// Mitsubishi GX Works2 project: Project   PLC: FX3G

// global labels: Global1
VAR_GLOBAL
  startDay AT X007 : BOOL;
  stillOpen AT Y007 : BOOL;
  Click_X5 AT X005 : BOOL;
  Analog_Output AT D8282 : INT;
  Analog_Input1 AT D8280 : INT;
  raspberryInentory AT D1111 : REAL;
  lemonInentory AT D2222 : REAL;
  stabilizerInentory AT D3333 : REAL;
  gummyBearsInentory AT D4444 : REAL;
  raspberryIceCreamRegular : REAL;
  raspberryIceCreamTreat : REAL;
  lemonIceCreamRegular : REAL;
  lemonIceCreamTreat : REAL;
  raspberryIceCreamContainer : REAL;
  lemonIceCreamContainer : REAL;
  coolingContainerRasp : REAL;
  coolingContainerLemon : REAL;
  mixContainer : REAL;
  startIceCreaming AT X001 : BOOL;
END_VAR
VAR_GLOBAL CONSTANT
  normalization : REAL := E400;
  ifLessThan10 : REAL := E10;
END_VAR
VAR_GLOBAL
  isRegular AT M1 : BOOL;
  isTreat AT M2 : BOOL;
END_VAR
VAR_GLOBAL CONSTANT
  rasbNeededRegular : REAL := E280.0;
  lemonNeededRegular : REAL := E455.0;
  stabNeededRegular : REAL := E105.0;
  bearNeededRegular : REAL := E28.0;
  rasbNeededTreat : REAL := E385.0;
  lemonNeededTreat : REAL := E665.0;
  stabNeededTreat : REAL := E210.0;
  bearNeededTreat : REAL := E70.0;
END_VAR
VAR_GLOBAL
  isRegPossible AT M3 : BOOL;
  isTreatPossible AT M4 : BOOL;
  FinishRegularToday AT M15 : BOOL;
  FinishTreatToday AT M16 : BOOL;
  StillPossible AT M50 : BOOL;
  FisrtStageIceCreamingReg AT M5 : BOOL;
  FisrtStageIceCreamingTreat AT M6 : BOOL;
  iceCreamDuration AT Y000 : BOOL;
  TimeCoil AT TC1 : BOOL;
  FiveSec AT K50 : INT;
  TimerWhileIceCreaming AT TS1 : BOOL;
END_VAR
VAR_GLOBAL CONSTANT
  raspberryIceCreamAddReg : REAL := E350.0;
  lemonIceCreamAddReg : REAL := E490.0;
  raspberryIceCreamAddTreat : REAL := E560.0;
  lemonIceCreamAddTreat : REAL := E700.0;
END_VAR
VAR_GLOBAL
  Sen_10 AT X003 : BOOL;
  TransferIceCream AT X002 : BOOL;
  LightForCooling AT Y002 : BOOL;
  TimerWhileCooling AT TC2 : BOOL;
  EightSec AT K80 : INT;
  TimerWhileCoolings AT TS2 : BOOL;
  MixRegular AT M51 : BOOL;
  MixTreat AT M61 : BOOL;
  WhileMixing_1 AT Y005 : BOOL;
  M_46 AT M46 : BOOL;
  startBlink5 AT TC50 : BOOL;
  MixingRegular AT TC30 : BOOL;
  MixingReg AT K30 : INT;
  MixingTreat AT TC55 : BOOL;
  DoneMixingRegular AT TS30 : BOOL;
  DoneMixingTreat AT TS55 : BOOL;
  Blink AT K5 : INT;
  ifEnoughBearRegular AT M7 : BOOL;
  ifEnoughBearTreat AT M8 : BOOL;
  Y5_Blinking AT TS50 : BOOL;
  startBlink6 AT TC60 : BOOL;
  Y6_Blinking AT TS60 : BOOL;
  WhileMixing_2 AT Y006 : BOOL;
  Pack1gumigum AT X000 : BOOL;
  IndicatorForX0 AT M20 : BOOL;
  cc1 AT CC1 : BOOL;
  startPacking AT X004 : BOOL;
  FirstGumigumInPackage AT Y004 : BOOL;
  GumigumPackage AT CS1 : BOOL;
  CounterGummies_7 AT K7 : INT;
  stillPacking AT M80 : BOOL;
  NumOfGummygamPacks AT D8284 : REAL;
END_VAR
VAR_GLOBAL CONSTANT
  AddPack : REAL := E0.01;
  MulConst : REAL := E4000.0;
  bearsForReg : REAL := E28.0;
  bearsForTreat : REAL := E70.0;
END_VAR
VAR_GLOBAL
  storageContainer : REAL;
END_VAR
VAR_GLOBAL CONSTANT
  storageCounter : REAL := E1.0;
  regularAmount : REAL := E868;
  treatAmount : REAL := E1330;
  ifGreaterThan6 : REAL := E6;
  ifBetween0_5 : REAL := E5;
  reset : REAL := E0.0;
END_VAR
VAR_GLOBAL
  finishedIteration AT M100 : BOOL;
  ifDone AT M200 : BOOL;
END_VAR

// task Task_01 (event TRUE, interval 0, priority 31): POU_01

PROGRAM POU_01
(* structured ladder/FBD written out as ST: instructions are called as NAME(EN, inputs, outputs); _pN, _eN, _tN stand for wires *)
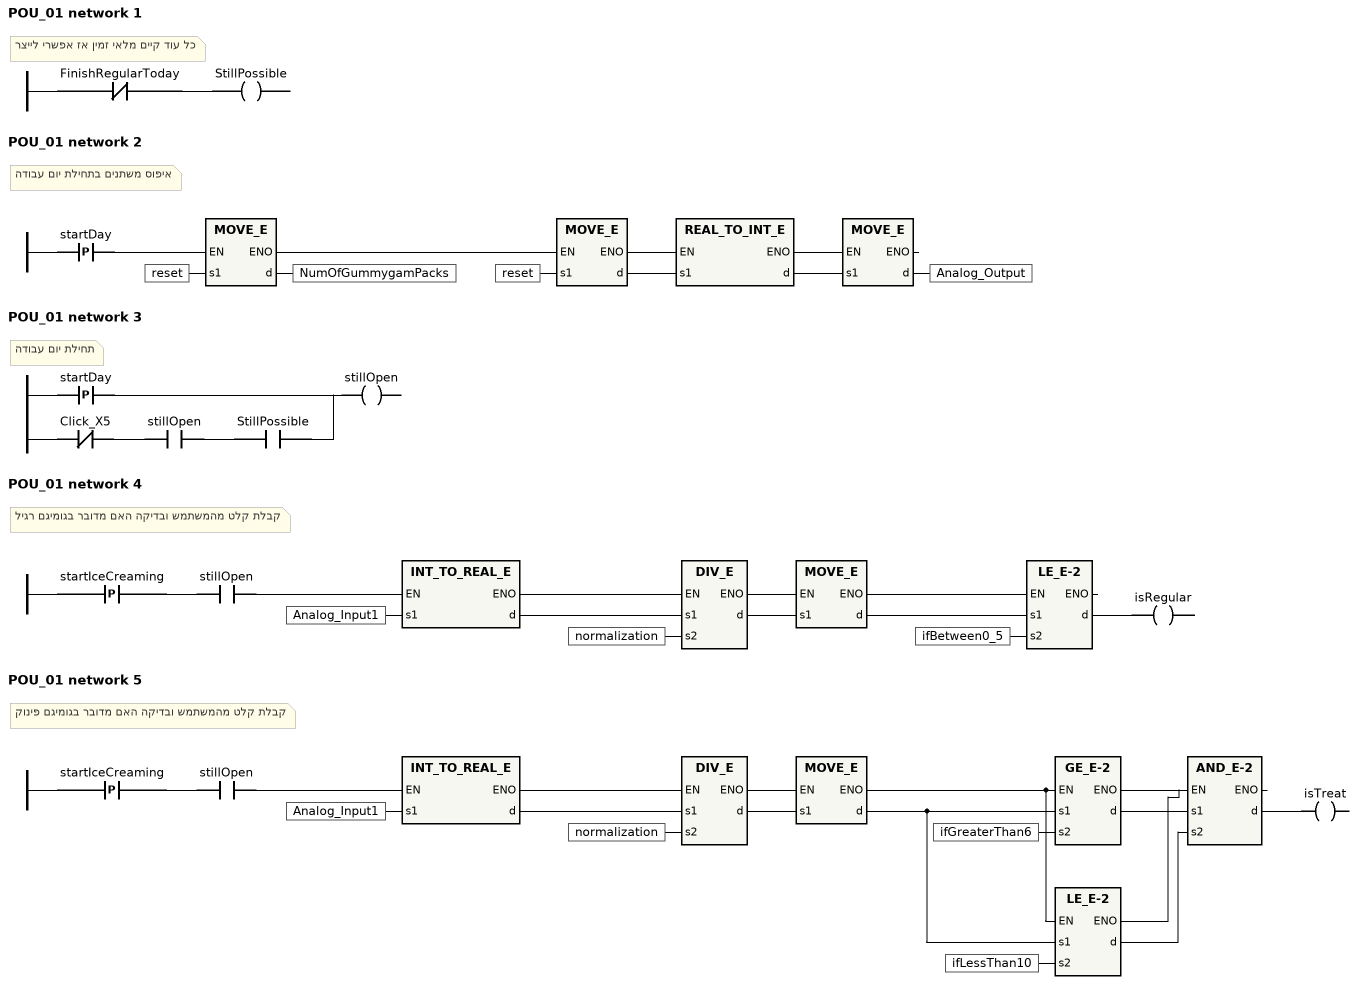
(* network 1 *)
(* כל עוד קיים מלאי זמין אז אפשרי לייצר *)
StillPossible := NOT FinishRegularToday;
(* network 2 *)
(* איפוס משתנים בתחילת יום עבודה *)
_e1 := MOVE_E(LDP(TRUE, startDay), reset, NumOfGummygamPacks);
_e3 := MOVE_E(_e1, reset, _t2);
_e5 := REAL_TO_INT_E(_e3, _t2, _t4);
MOVE_E(_e5, _t4, Analog_Output);
(* network 3 *)
(* תחילת יום עבודה *)
stillOpen := LDP(TRUE, startDay) OR (NOT Click_X5 AND stillOpen AND StillPossible);
(* network 4 *)
(* קבלת קלט מהמשתמש ובדיקה האם מדובר בגומיגם רגיל *)
_e2 := INT_TO_REAL_E(LDP(TRUE, startIceCreaming) AND stillOpen, Analog_Input1, _t1);
_e4 := DIV_E(_e2, _t1, normalization, _t3);
_e6 := MOVE_E(_e4, _t3, _t5);
LE_E(_e6, _t5, ifBetween0_5, _t7);
isRegular := _t7;
(* network 5 *)
(* קבלת קלט מהמשתמש ובדיקה האם מדובר בגומיגם פינוק *)
_e2 := INT_TO_REAL_E(LDP(TRUE, startIceCreaming) AND stillOpen, Analog_Input1, _t1);
_e4 := DIV_E(_e2, _t1, normalization, _t3);
_e6 := MOVE_E(_e4, _t3, _t5);
_e8 := GE_E(_e6, _t5, ifGreaterThan6, _t7);
_e10 := LE_E(_e6, _t5, ifLessThan10, _t9);
AND_E(_e8 OR _e10, _t7, _t9, _t11);
isTreat := _t11;
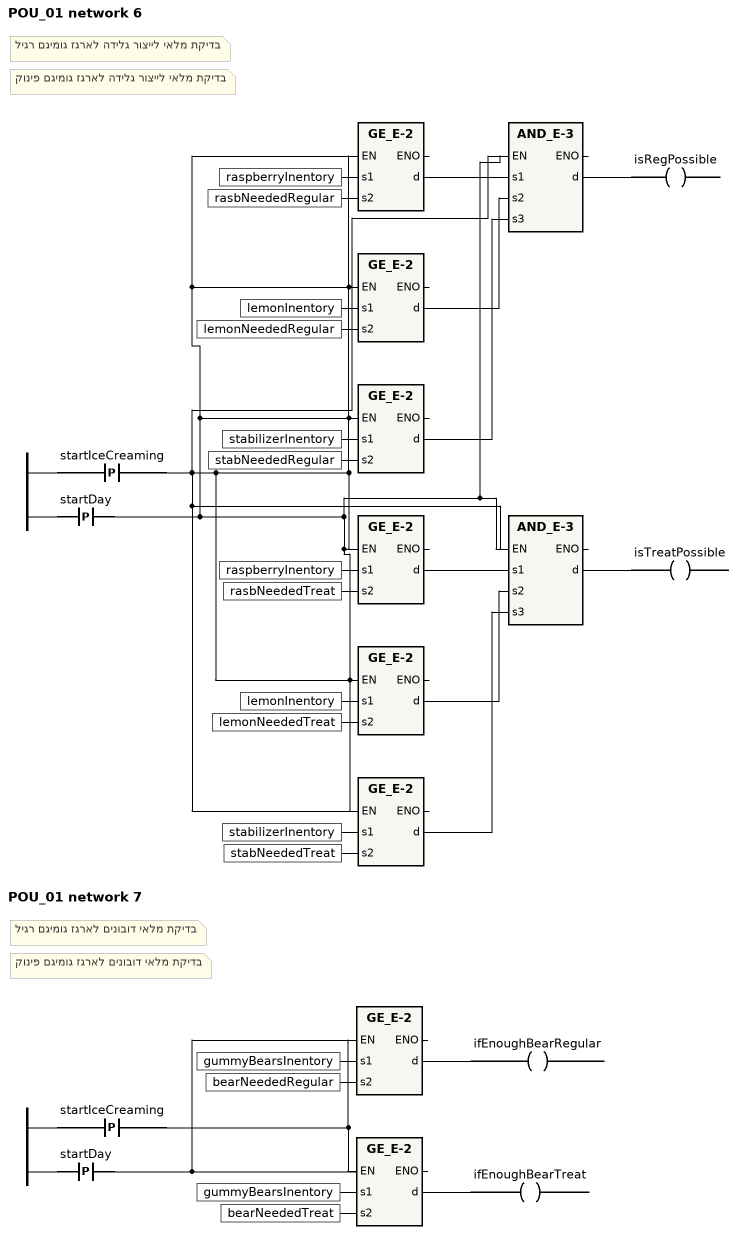
(* network 6 *)
(* בדיקת מלאי לייצור גלידה לארגז גומיגם רגיל *)
(* בדיקת מלאי לייצור גלידה לארגז גומיגם פינוק *)
_p1 := LDP(TRUE, startIceCreaming) OR LDP(TRUE, startDay);
GE_E(_p1, raspberryInentory, rasbNeededRegular, _t2);
GE_E(_p1, lemonInentory, lemonNeededRegular, _t3);
GE_E(_p1, stabilizerInentory, stabNeededRegular, _t4);
AND_E(_p1, _t2, _t3, _t4, _t5);
isRegPossible := _t5;
GE_E(_p1, raspberryInentory, rasbNeededTreat, _t6);
GE_E(_p1, lemonInentory, lemonNeededTreat, _t7);
GE_E(_p1, stabilizerInentory, stabNeededTreat, _t8);
AND_E(_p1, _t6, _t7, _t8, _t9);
isTreatPossible := _t9;
(* network 7 *)
(* בדיקת מלאי דובונים לארגז גומיגם רגיל *)
(* בדיקת מלאי דובונים לארגז גומיגם פינוק *)
_p1 := LDP(TRUE, startIceCreaming) OR LDP(TRUE, startDay);
GE_E(_p1, gummyBearsInentory, bearNeededRegular, _t2);
ifEnoughBearRegular := _t2;
GE_E(_p1, gummyBearsInentory, bearNeededTreat, _t3);
ifEnoughBearTreat := _t3;
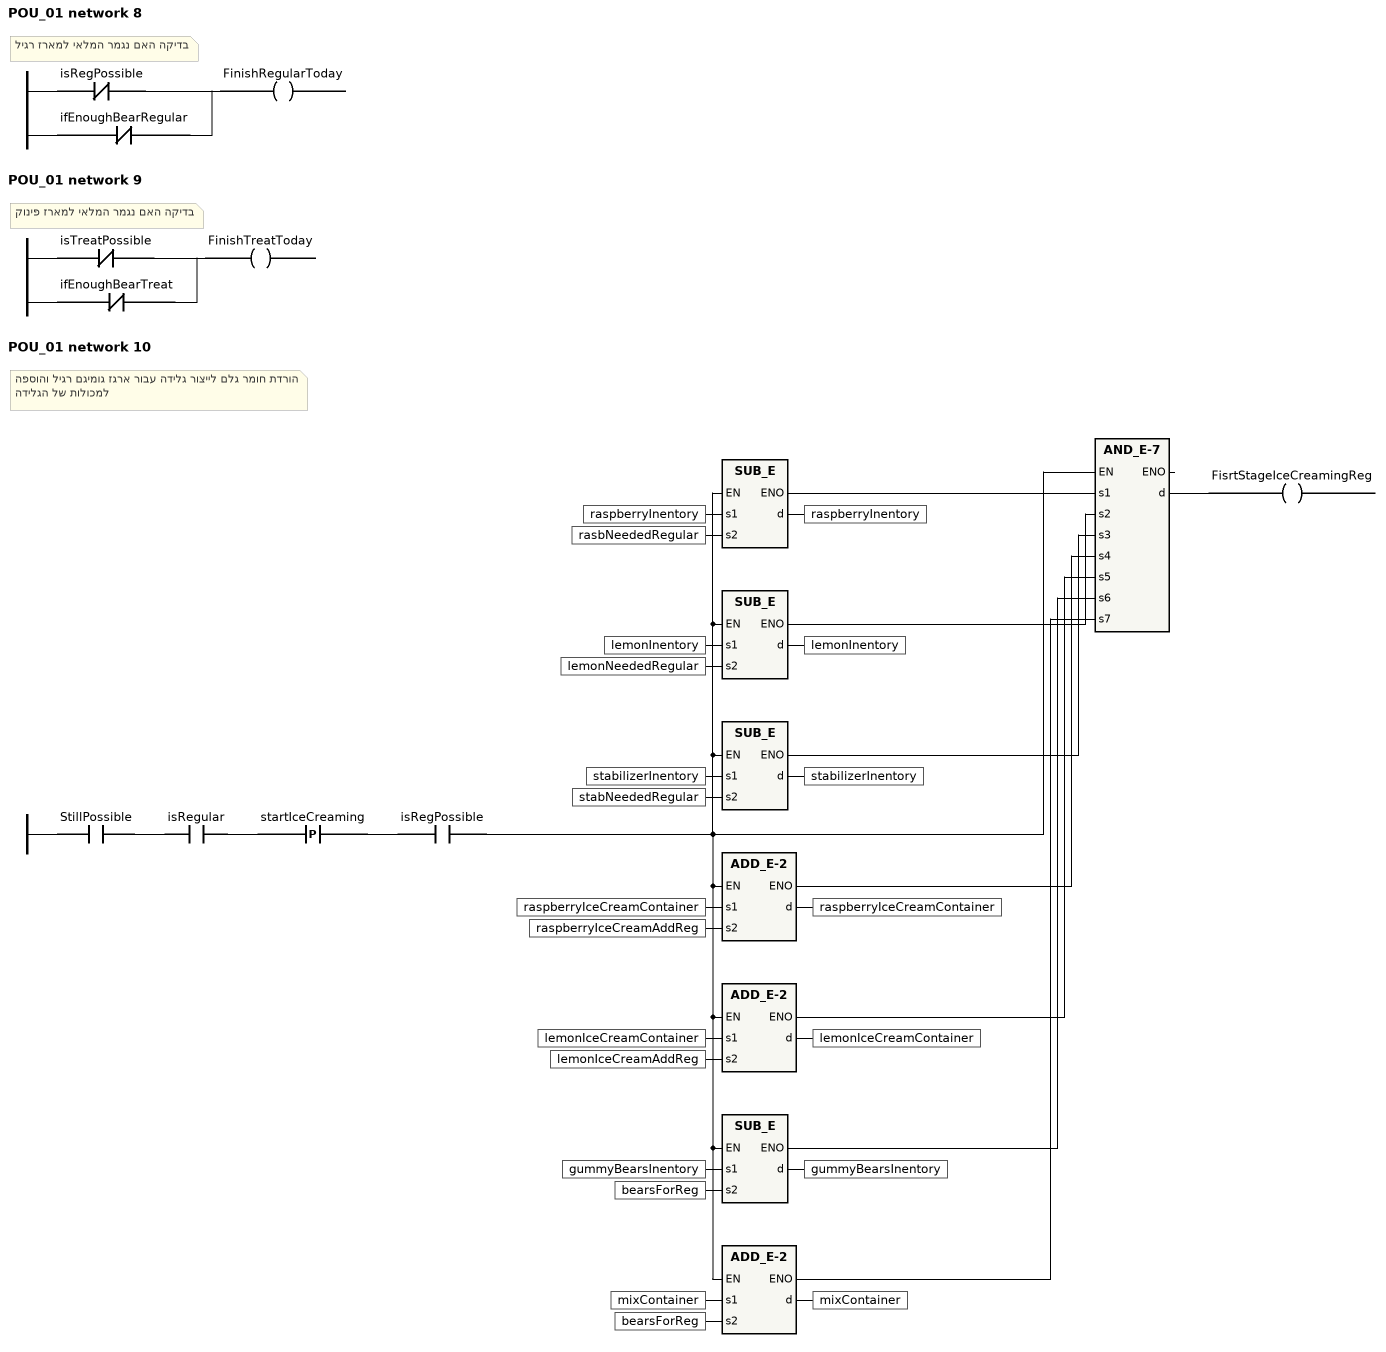
(* network 8 *)
(* בדיקה האם נגמר המלאי למארז רגיל *)
FinishRegularToday := (NOT isRegPossible) OR (NOT ifEnoughBearRegular);
(* network 9 *)
(* בדיקה האם נגמר המלאי למארז פינוק *)
FinishTreatToday := (NOT isTreatPossible) OR (NOT ifEnoughBearTreat);
(* network 10 *)
(* הורדת חומר גלם לייצור גלידה עבור ארגז גומיגם רגיל והוספה למכולות של הגלידה *)
_p1 := StillPossible AND isRegular AND LDP(TRUE, startIceCreaming) AND isRegPossible;
_e2 := SUB_E(_p1, raspberryInentory, rasbNeededRegular, raspberryInentory);
_e3 := SUB_E(_p1, lemonInentory, lemonNeededRegular, lemonInentory);
_e4 := SUB_E(_p1, stabilizerInentory, stabNeededRegular, stabilizerInentory);
_e5 := ADD_E(_p1, raspberryIceCreamContainer, raspberryIceCreamAddReg, raspberryIceCreamContainer);
_e6 := ADD_E(_p1, lemonIceCreamContainer, lemonIceCreamAddReg, lemonIceCreamContainer);
_e7 := SUB_E(_p1, gummyBearsInentory, bearsForReg, gummyBearsInentory);
_e8 := ADD_E(_p1, mixContainer, bearsForReg, mixContainer);
AND_E(_p1, _e2, _e3, _e4, _e5, _e6, _e7, _e8, _t9);
FisrtStageIceCreamingReg := _t9;
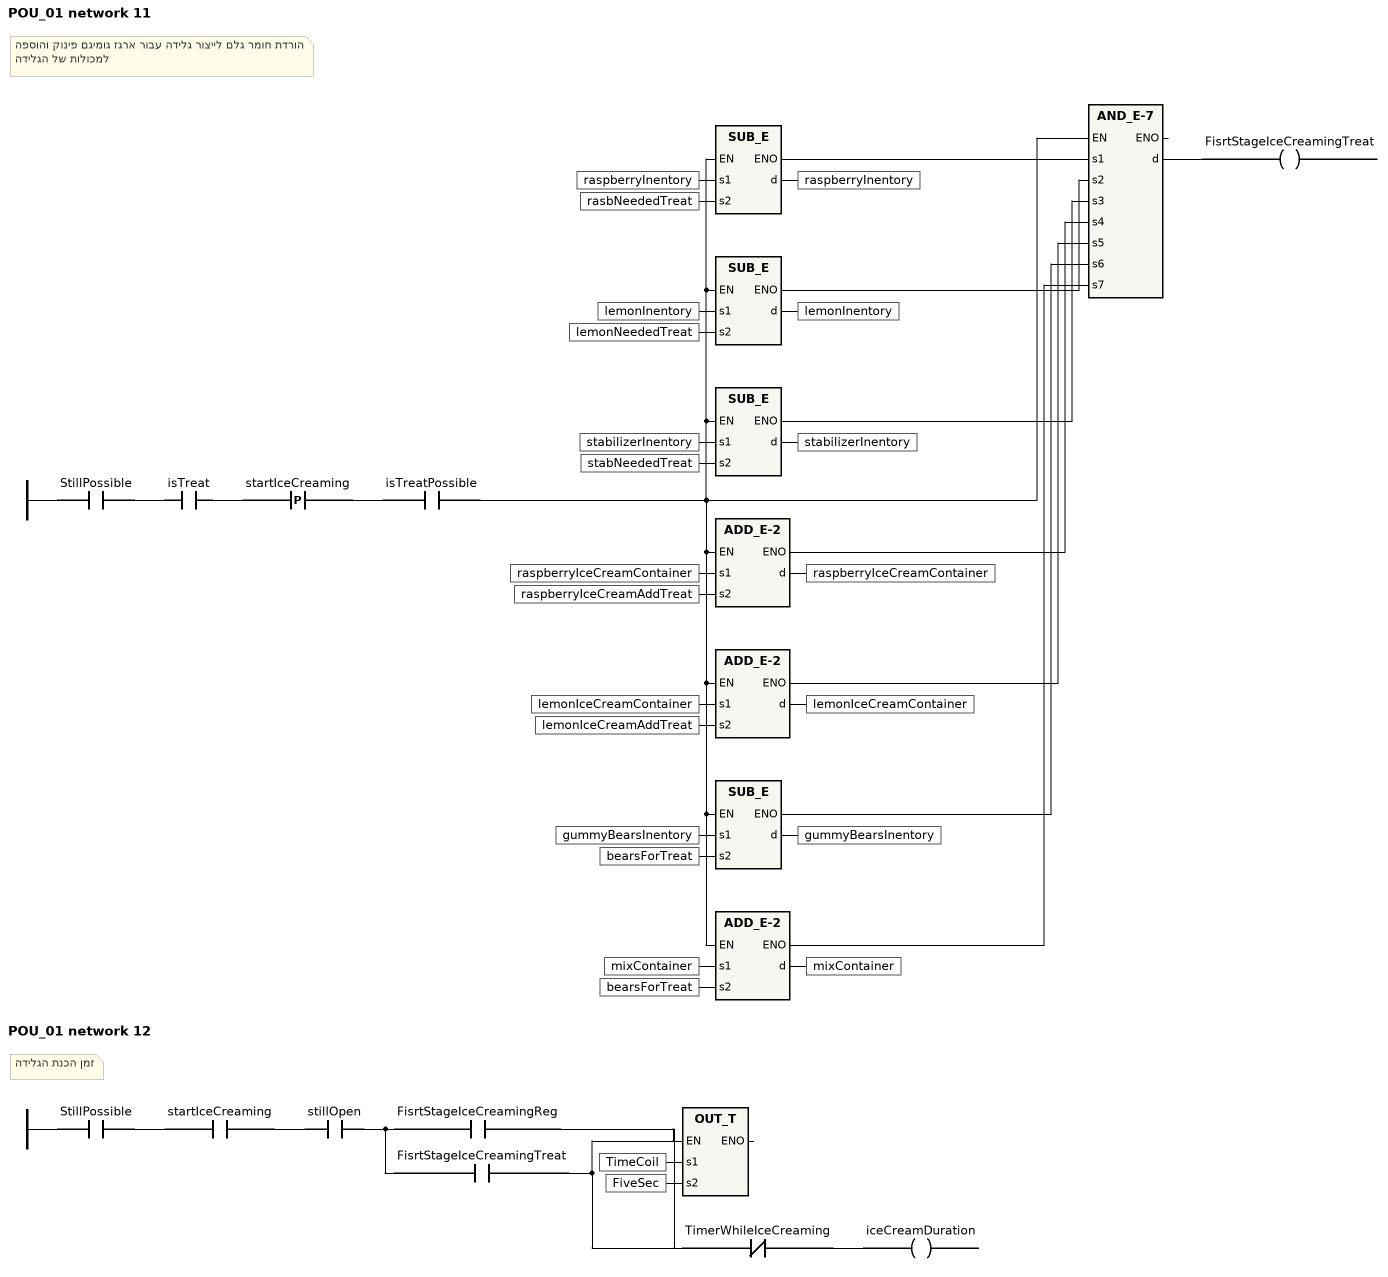
(* network 11 *)
(* הורדת חומר גלם לייצור גלידה עבור ארגז גומיגם פינוק והוספה למכולות של הגלידה *)
_p1 := StillPossible AND isTreat AND LDP(TRUE, startIceCreaming) AND isTreatPossible;
_e2 := SUB_E(_p1, raspberryInentory, rasbNeededTreat, raspberryInentory);
_e3 := SUB_E(_p1, lemonInentory, lemonNeededTreat, lemonInentory);
_e4 := SUB_E(_p1, stabilizerInentory, stabNeededTreat, stabilizerInentory);
_e5 := ADD_E(_p1, raspberryIceCreamContainer, raspberryIceCreamAddTreat, raspberryIceCreamContainer);
_e6 := ADD_E(_p1, lemonIceCreamContainer, lemonIceCreamAddTreat, lemonIceCreamContainer);
_e7 := SUB_E(_p1, gummyBearsInentory, bearsForTreat, gummyBearsInentory);
_e8 := ADD_E(_p1, mixContainer, bearsForTreat, mixContainer);
AND_E(_p1, _e2, _e3, _e4, _e5, _e6, _e7, _e8, _t9);
FisrtStageIceCreamingTreat := _t9;
(* network 12 *)
(* זמן הכנת הגלידה *)
_p1 := StillPossible AND startIceCreaming AND stillOpen;
_p2 := (_p1 AND FisrtStageIceCreamingReg) OR (_p1 AND FisrtStageIceCreamingTreat);
iceCreamDuration := _p2 AND NOT TimerWhileIceCreaming;
OUT_T(_p2, TimeCoil, FiveSec);
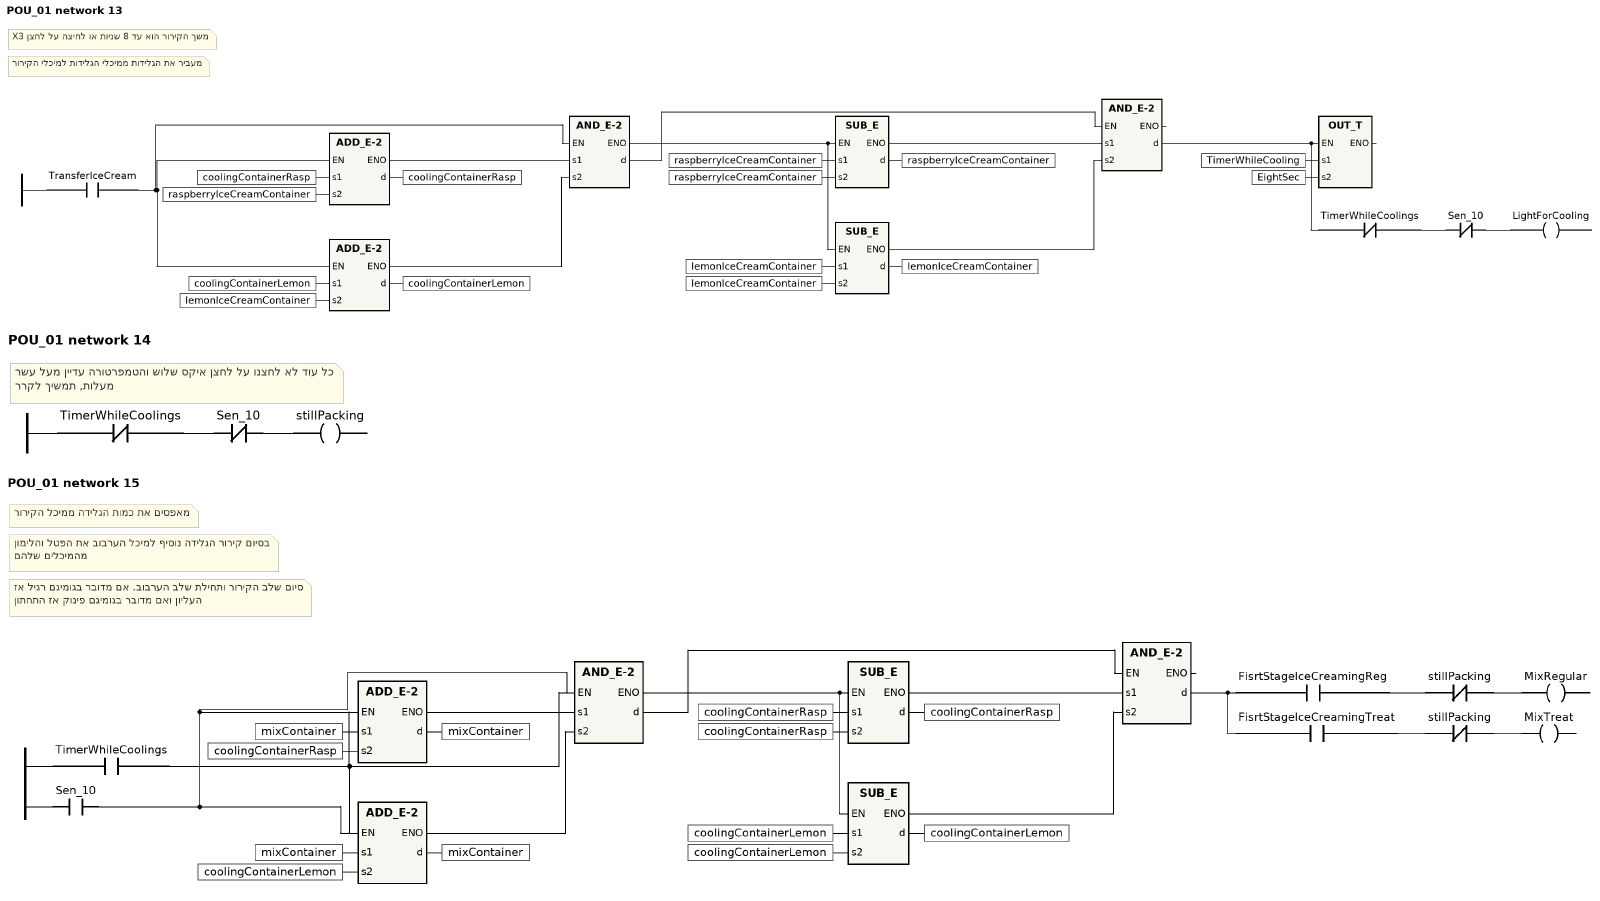
(* network 13 *)
(* משך הקירור הוא עד 8 שניות או לחיצה על לחצן X3 *)
(* מעביר את הגלידות ממיכלי הגלידות למיכלי הקירור *)
_e1 := ADD_E(TransferIceCream, coolingContainerRasp, raspberryIceCreamContainer, coolingContainerRasp);
_e2 := ADD_E(TransferIceCream, coolingContainerLemon, lemonIceCreamContainer, coolingContainerLemon);
_e4 := AND_E(TransferIceCream, _e1, _e2, _t3);
_e5 := SUB_E(_e4, raspberryIceCreamContainer, raspberryIceCreamContainer, raspberryIceCreamContainer);
_e6 := SUB_E(_e4, lemonIceCreamContainer, lemonIceCreamContainer, lemonIceCreamContainer);
AND_E(_t3, _e5, _e6, _t7);
LightForCooling := _t7 AND NOT TimerWhileCoolings AND NOT Sen_10;
OUT_T(_t7, TimerWhileCooling, EightSec);
(* network 14 *)
(* כל עוד לא לחצנו על לחצן איקס שלוש והטמפרטורה עדיין מעל עשר מעלות, תמשיך לקרר *)
stillPacking := NOT TimerWhileCoolings AND NOT Sen_10;
(* network 15 *)
(* מאפסים את כמות הגלידה ממיכל הקירור *)
(* בסיום קירור הגלידה נוסיף למיכל הערבוב את הפטל והלימון מהמיכלים שלהם *)
(* סיום שלב הקירור ותחילת שלב הערבוב. אם מדובר בגומיגם רגיל אז העליון ואם מדובר בגומיגם פינוק אז התחתון *)
_p1 := TimerWhileCoolings OR Sen_10;
_e2 := ADD_E(_p1, mixContainer, coolingContainerRasp, mixContainer);
_e3 := ADD_E(_p1, mixContainer, coolingContainerLemon, mixContainer);
_e5 := AND_E(_p1, _e2, _e3, _t4);
_e6 := SUB_E(_e5, coolingContainerRasp, coolingContainerRasp, coolingContainerRasp);
_e7 := SUB_E(_e5, coolingContainerLemon, coolingContainerLemon, coolingContainerLemon);
AND_E(_t4, _e6, _e7, _t8);
MixRegular := _t8 AND FisrtStageIceCreamingReg AND NOT stillPacking;
MixTreat := _t8 AND FisrtStageIceCreamingTreat AND NOT stillPacking;
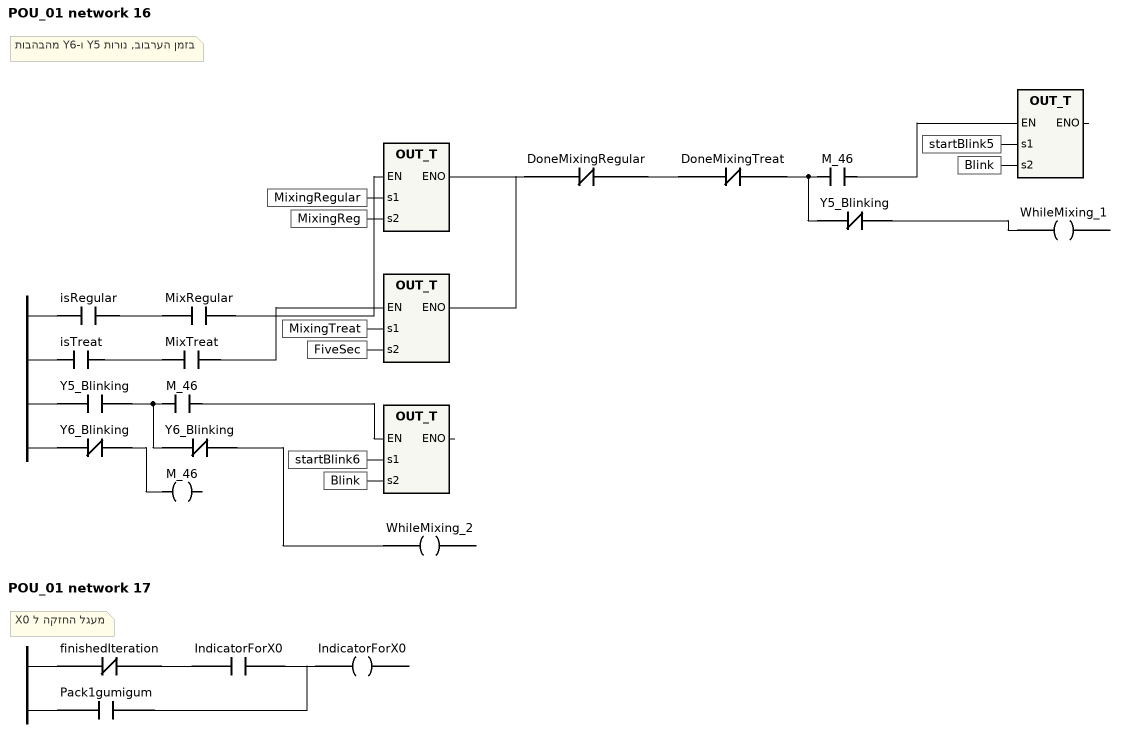
(* network 16 *)
(* בזמן הערבוב, נורות Y5 ו-Y6 מהבהבות *)
_e1 := OUT_T(isRegular AND MixRegular, MixingRegular, MixingReg);
_e2 := OUT_T(isTreat AND MixTreat, MixingTreat, FiveSec);
_p3 := ((_e1 OR _e2) AND NOT DoneMixingRegular) AND NOT DoneMixingTreat;
OUT_T(_p3 AND M_46, startBlink5, Blink);
WhileMixing_1 := _p3 AND NOT Y5_Blinking;
OUT_T(Y5_Blinking AND M_46, startBlink6, Blink);
WhileMixing_2 := Y5_Blinking AND NOT Y6_Blinking;
M_46 := NOT Y6_Blinking;
(* network 17 *)
(* מעגל החזקה ל X0 *)
IndicatorForX0 := (NOT finishedIteration AND IndicatorForX0) OR Pack1gumigum;
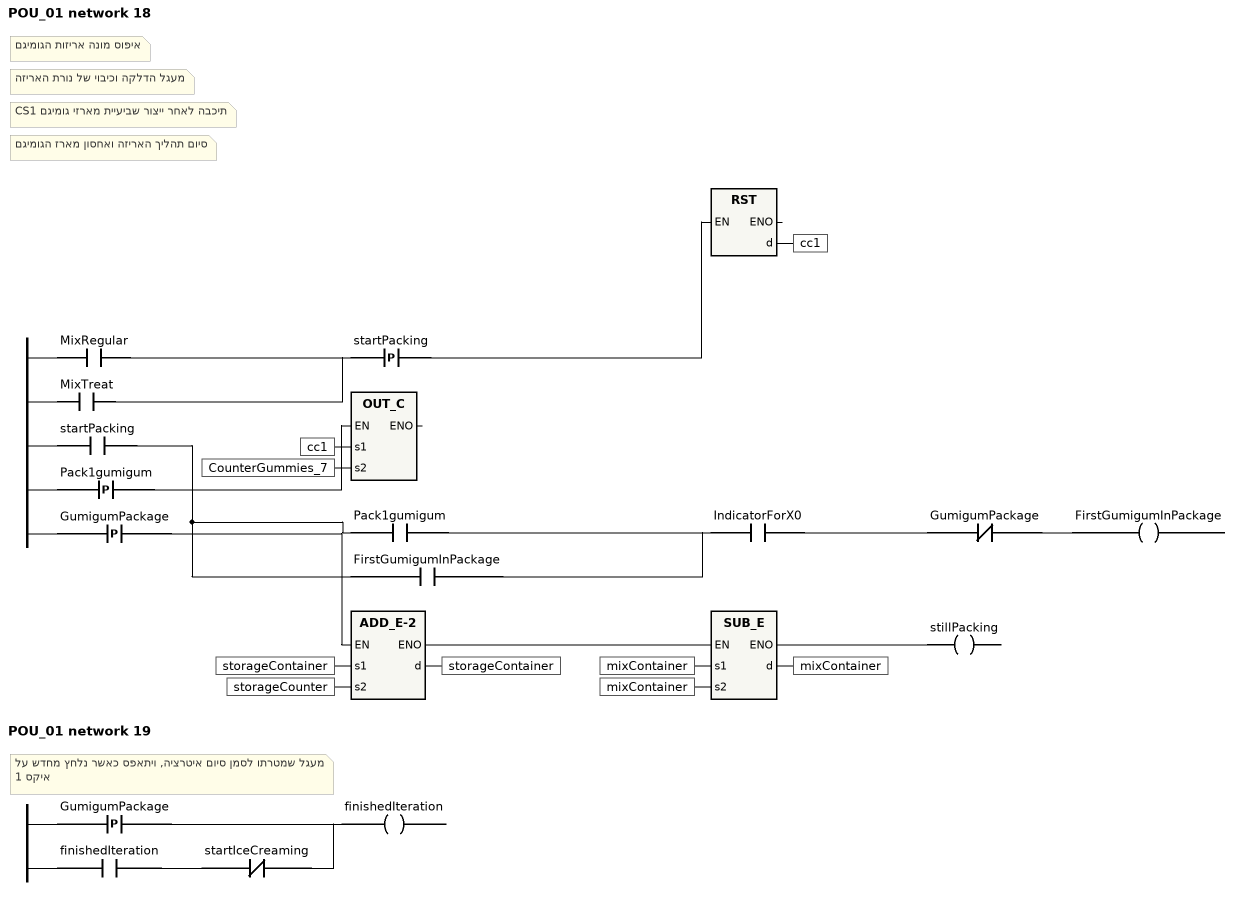
(* network 18 *)
(* איפוס מונה אריזות הגומיגם *)
(* מעגל הדלקה וכיבוי של נורת האריזה *)
(* CS1 תיכבה לאחר ייצור שביעיית מארזי גומיגם *)
(* סיום תהליך האריזה ואחסון מארז הגומיגם *)
RST((MixRegular OR MixTreat) AND LDP(TRUE, startPacking), cc1);
FirstGumigumInPackage := (((startPacking AND Pack1gumigum) OR (startPacking AND FirstGumigumInPackage)) AND IndicatorForX0) AND NOT GumigumPackage;
OUT_C(LDP(TRUE, Pack1gumigum), cc1, CounterGummies_7);
_e1 := ADD_E(LDP(TRUE, GumigumPackage), storageContainer, storageCounter, storageContainer);
_e2 := SUB_E(_e1, mixContainer, mixContainer, mixContainer);
stillPacking := _e2;
(* network 19 *)
(* מעגל שמטרתו לסמן סיום איטרציה, ויתאפס כאשר נלחץ מחדש על איקס 1 *)
finishedIteration := LDP(TRUE, GumigumPackage) OR (finishedIteration AND NOT startIceCreaming);
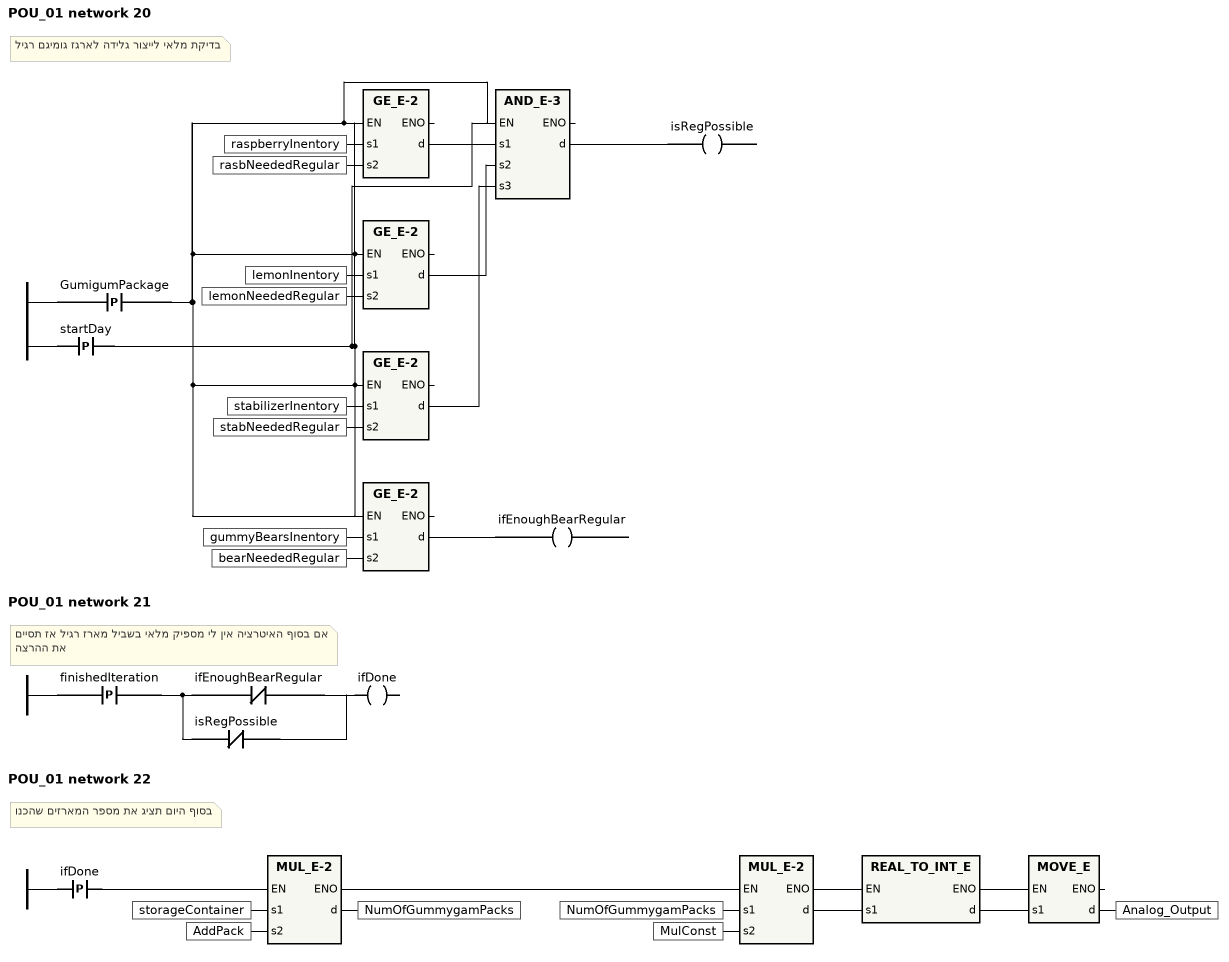
(* network 20 *)
(* בדיקת מלאי לייצור גלידה לארגז גומיגם רגיל *)
_p1 := LDP(TRUE, GumigumPackage) OR LDP(TRUE, startDay);
GE_E(_p1, raspberryInentory, rasbNeededRegular, _t2);
GE_E(_p1, lemonInentory, lemonNeededRegular, _t3);
GE_E(_p1, stabilizerInentory, stabNeededRegular, _t4);
AND_E(_p1, _t2, _t3, _t4, _t5);
isRegPossible := _t5;
GE_E(_p1, gummyBearsInentory, bearNeededRegular, _t6);
ifEnoughBearRegular := _t6;
(* network 21 *)
(* אם בסוף האיטרציה אין לי מספיק מלאי בשביל מארז רגיל אז תסיים את ההרצה *)
_p1 := LDP(TRUE, finishedIteration);
ifDone := (_p1 AND NOT ifEnoughBearRegular) OR (_p1 AND NOT isRegPossible);
(* network 22 *)
(* בסוף היום תציג את מספר המארזים שהכנו *)
_e1 := MUL_E(LDP(TRUE, ifDone), storageContainer, AddPack, NumOfGummygamPacks);
_e3 := MUL_E(_e1, NumOfGummygamPacks, MulConst, _t2);
_e5 := REAL_TO_INT_E(_e3, _t2, _t4);
MOVE_E(_e5, _t4, Analog_Output);
END_PROGRAM
